(* CODESYS project Alert and Gif.ecp

Project tree, tasks and I/O mapping:
  PFC200_CS_2ETH_RS : 750-8212 PFC200 2ETH RS, WAGO, order no. 0750-8212, version 5.13.2.22
    application Application
      libraries: 
      task PLC_Task (cyclic, interval t#10ms, priority 14) calls PLC_PRG
      task VISU_TASK (cyclic, interval 100 ms, priority 15) calls VisuElems.Visu_Prg
      program PLC_PRG [ST]
      visualisation Visualization
    Common.PCI
    Kbus : Kbus, WAGO, version 1.4.0.2
        unmapped channels: K-BUS diagnostics
    MODBUS
      MODBUS : MODBUS, WAGO, order no. n/a, version 1.1.1.15
    Serial
      COM1 : COM1, WAGO, version 0.0.0.19
  TP600_10_1_1280x800_PIO3_CP : TP600 10.1 1280x800 PIO3 CP , WAGO, order no. 0762-5304, version 5.13.2.22
    application Application
      libraries: 
      task VISU_TASK (cyclic, interval 100 ms, priority 15) calls VisuElems.Visu_Prg
      task PLC_Task (cyclic, interval t#50ms, priority 15) calls PLC_PRG
      program PLC_PRG [ST]
      visualisation Visualization
    MODBUS
      MODBUS : MODBUS, WAGO, order no. n/a, version 1.1.1.15
    CANbus
    Common.PCI
    TP600_Onboard_IO : TP600 Onboard IO, WAGO, version 0.0.1.2
        unmapped channels: _IN, _OUT
    Serial
      COM1 : COM1, WAGO, version 0.0.0.19
  libraries: VisuSymbols, 3.5.10.0 (System); WagoVisuIcons, 1.0.1.0 (WAGO)
  text list GlobalTextList
*)

// PFC200_CS_2ETH_RS/Application/PLC_PRG
PROGRAM PLC_PRG
VAR
	xtest:BOOL;
END_VAR

END_PROGRAM

// TP600_10_1_1280x800_PIO3_CP/Application/PLC_PRG
PROGRAM PLC_PRG
VAR
	xAlert:BOOL;
	xAlert2:BOOL;
END_VAR

END_PROGRAM

// PFC200_CS_2ETH_RS/Application/Visualization
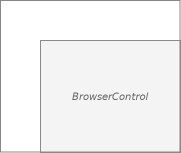
VISUALIZATION Visualization  // 181x153
    BrowserControl (40,40 141x113)
        p3734058945: 'http://192.168.1.212/Sound.html'
        p2179181546: PLC_PRG.xtest
END_VISUALIZATION

// TP600_10_1_1280x800_PIO3_CP/Application/Visualization
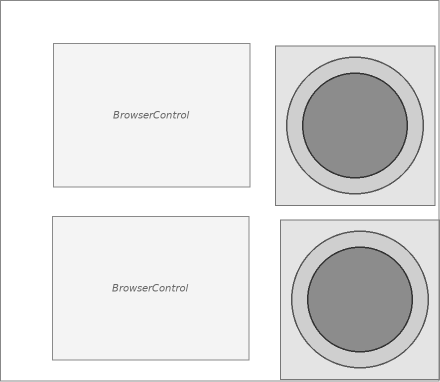
VISUALIZATION Visualization  // 440x382
    BrowserControl (53,43 197x144)
        p2179181546: PLC_PRG.xAlert
        p3734058945: 'http://192.168.1.173/Sound.html'
    PushSwitchLed (275,43 160x165), variable: PLC_PRG.xAlert, behaviour: TAP, style: Switch-PushSwitchLed-Gray
    BrowserControl (52,216 197x144)
        p2179181546: PLC_PRG.xAlert2
        p3734058945: 'http://192.168.1.173/Sound2.html'
    PushSwitchLed (280,217 160x165), variable: PLC_PRG.xAlert2, behaviour: TAP, style: Switch-PushSwitchLed-Gray
END_VISUALIZATION
